Staubli VAL3: insertItem.pgx

public program insertItem(num& x_nIndexCopy, num x_nIndexPaste)
  local num l_nLastType
  local point l_pPoint
  local num l_nType
begin
  //
  // use to add more elements from the typical one
  //
  // insert all the field
  //
  l_pPoint=pEditPoint.tData[x_nIndexCopy].pPoint
  l_nLastType=pEditPoint.tData[x_nIndexCopy].nType
  if l_nLastType==0
    l_nType=0
  elseIf l_nLastType==2 or l_nLastType==1
    l_nType=2
  endIf
  insert(pEditPoint.tData[x_nIndexPaste])
  // set IT - link it
  link(pEditPoint.tData[x_nIndexPaste].pPoint,pEditPoint.fFrame)
  link(pEditPoint.tData[x_nIndexPaste].pCircle,pEditPoint.fFrame)
  pEditPoint.tData[x_nIndexPaste].pPoint.trsf=l_pPoint.trsf
  // set IT
  pEditPoint.tData[x_nIndexPaste].nType=l_nType
end
